// TwinCAT 3 PLC project PLCstudent
// ProgramVersion: 3.1.4026.19
// libraries:
//   Tc2_Standard, * (Beckhoff Automation GmbH)
//   Tc2_System, * (Beckhoff Automation GmbH)
// project tree:
//   GVLs/ GVL.TcGVL
//   / PlcTask.TcTTO
//   POUs/ FunktionBlockDiagram.TcPOU, MAIN.TcPOU
// real-time tasks:
//   TASK PlcTask: cycle T#10ms, priority 20, ADS port 350
//   TASK PlcTask1: cycle T#10ms, priority 21, ADS port 351
// variable links:
//   PLCsim/PLCsim Instance <-> PLCstudent/PLCstudent Instance
//     PlcTask Inputs/GVL.isStatusText <-> PlcTask Outputs/GVL.qsStatusText
//     PlcTask Inputs/GVL.iwPumpSpeed <-> PlcTask Outputs/GVL.qwPumpSpeed
//     PlcTask Outputs/GVL.qwActualLevel <-> PlcTask Inputs/GVL.iwActualLevel

CONFIGURATION PLCstudent
    RESOURCE PLC ON TwinCAT3
        TASK PlcTask(INTERVAL := T#10ms, PRIORITY := 20);
        PROGRAM MAIN WITH PlcTask : MAIN;
    END_RESOURCE
END_CONFIGURATION

// ---- GVLs/GVL.TcGVL
{attribute 'qualified_only'}
VAR_GLOBAL

	qwPumpSpeed   		AT%Q* :  WORD; 	// Speed of the flow into the tank 0 - 100%
										// 40% slowly drain 50% stand still 60% filling
										

	qsStatusText 		AT%Q* : STRING := 'Test text'; // Text on the info display
	
	iwActualLevel 		AT%I* : WORD;  	// Level in the tank	
	
END_VAR

// ---- POUs/MAIN.TcPOU
VAR
    iActualLevelInt : INT;    // 转换后的水位整数
    iControlOutput  : INT;    // 计算出的控制输出结果
    iKp             : INT := 50; // 比例增益，初始为 10
END_VAR


// -------------------------------------------------------------------------
// TASK 2: Simple Proportional (P) Controller
// Formula: Speed = (Set - Is) * Kp
// -------------------------------------------------------------------------

// Step 1: Convert WORD to INT to allow negative results in subtraction (Requirement: OBS!)
iActualLevelInt := WORD_TO_INT(GVL.iwActualLevel);

// Step 2: Calculate difference from Setpoint (50) and multiply by Gain (Kp)
iControlOutput := (50 - iActualLevelInt) * iKp;

// Step 3: Handle negative values and assign to Pump Speed (Requirement: SEL function logic)
// If level > 50, calculation is negative. Pump speed cannot be negative.
IF iControlOutput < 0 THEN
    GVL.qwPumpSpeed := 0;
ELSE
    // Convert back to WORD for the global variable
    GVL.qwPumpSpeed := INT_TO_WORD(iControlOutput);
END_IF;


// -------------------------------------------------------------------------
// TASK 1: Level Indication and Status Text
// Using ranges to prevent flickering/jitter on the display
// -------------------------------------------------------------------------

IF GVL.iwActualLevel < 40 THEN
    // Below 40%: Low level status
    GVL.qsStatusText := 'Low level';
    
ELSIF GVL.iwActualLevel >= 40 AND GVL.iwActualLevel <= 60 THEN
    // Between 40% and 60%: Normal operating range
    GVL.qsStatusText := 'Normal level';
    
ELSE
    // Above 60%: High level status
    GVL.qsStatusText := 'High level';
END_IF;

// -------------------------------------------------------------------------
// TASK 3: Call Function Block Diagram
// -------------------------------------------------------------------------
FunktionBlockDiagram();

// ---- POUs/FunktionBlockDiagram.TcPOU
PROGRAM FunktionBlockDiagram
VAR
	
END_VAR

END_PROGRAM
